INTERFACE ICommand

METHOD Refresh
END_METHOD

END_INTERFACE

(* stored: Version 1.1.0.1, ProductVersion 3.1.4022.10
   Itf ICommand: Id {9dc6c476-c433-07d6-317f-3d274872f03c}
   Method Refresh: Id {b0863e7e-d159-0a36-1b9e-7efd24b9bd48} *)
